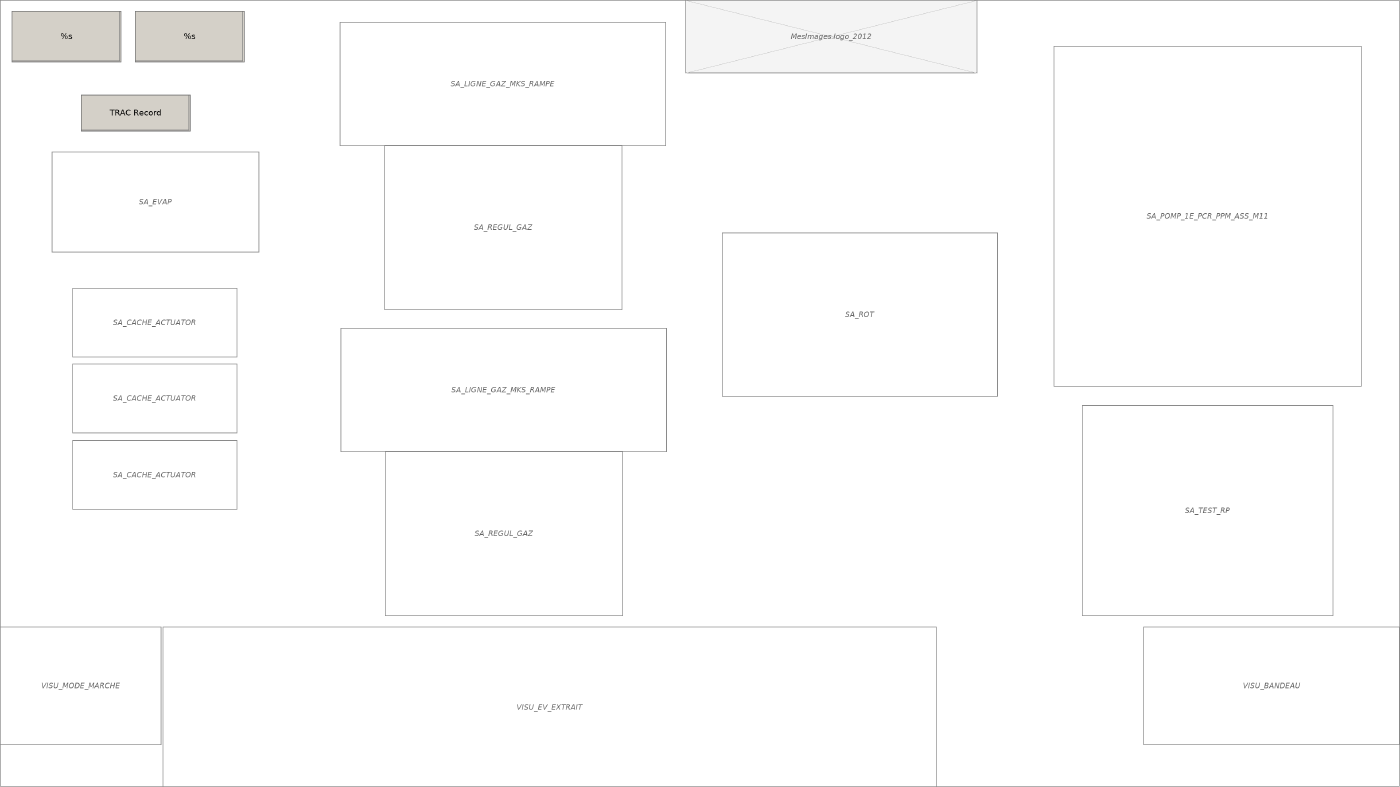
VISUALIZATION VISU_SA  // 1920x1080, background image fond_blanc_1280_1024
    Frame (223,860 1061x221)
        shows VISU_EV_EXTRAIT()
    Frame (1568,860 352x162)
        shows VISU_BANDEAU(m_Input_MACHINE := Global_Variables.MACHINE)
    Frame (0,860 221x162)
        shows VISU_MODE_MARCHE(m_Input_MACHINE := .MACHINE)
    Frame (71,208 284x138)
        shows SA_EVAP(m_Input_Crucible := PRG_EVAP.CRUCIBLE1, m_Input_Sweep := PRG_EVAP.SWEEP1)
    Frame (99,395 226x95)
        shows SA_CACHE_ACTUATOR(m_Input_CACHE := PRG_EVAP.CC11, m_Input_PRM_Forcage := PRG_EVAP.PRM_Forcage_Cache_Source1)
    Frame (466,30 447x170)
        shows SA_LIGNE_GAZ_MKS_RAMPE(m_Input_Ligne := PRG_GAZ.LIGNE_GAZ[1], m_Input_Machine := MACHINE, m_Input_DG := .PRG_GAZ.DG[1], m_Input_UserRight := PRG_USER.ACTU_USER.FONCTION_SA, m_Input_NumTextList := 11)
    Frame (99,499 226x95)
        shows SA_CACHE_ACTUATOR(m_Input_CACHE := PRG_EVAP.CC12, m_Input_PRM_Forcage := PRG_EVAP.PRM_Forcage_Cache_Source2)
    Frame (990,319 378x225)
        shows SA_ROT(m_Input_ROT := PRG_MOUVEMENT_PS.ROTATION_PS, m_Input_PRG := PRG_MOUVEMENT_PS)
    Frame (99,604 226x95)
        shows SA_CACHE_ACTUATOR(m_Input_CACHE := PRG_EVAP.CC13, m_Input_PRM_Forcage := PRG_EVAP.PRM_Forcage_Cache_Source3)
    Button (16,15 150x70), "%s", text list: 'TextList_Navigation', text index: 0
        OnMouseClick: change screen: SYN_POMPAGE
    Button (185,15 150x70), "%s", text list: 'TextList_Navigation', text index: 1
        OnMouseClick: change screen: SYN_PROC
    Frame (527,199 326x226)
        shows SA_REGUL_GAZ(m_Input_REGULATION := PRG_GAZ.REGULATION_GAZ_L1, m_Input_MACHINE := .MACHINE)
    Frame (528,619 326x226)
        shows SA_REGUL_GAZ(m_Input_REGULATION := PRG_GAZ.REGULATION_GAZ_L2, m_Input_MACHINE := .MACHINE)
    Frame (1484,556 344x289)
        shows SA_TEST_RP(m_Input_Operation := PRG_POMPAGE.POMPAGE.OP_Test_RP, m_Input_Pression := PRG_POMPAGE.POMPAGE.PRM_Pr_test, m_Input_Duree := PRG_POMPAGE.POMPAGE.PRM_Tim_test, m_Input_Volume := PRG_POMPAGE.POMPAGE.CONF_Volume_Enceinte, m_Input_Co_Stop := PRG_POMPAGE.POMPAGE.CO_Stop_Test_RP, m_Input_Timer := PRG_POMPAGE.POMPAGE.TIMER_attente_test.ET, m_Input_Result := PRG_POMPAGE.POMPAGE.VAR_Indicateur_Test)
    Frame (1445,63 422x467)
        shows SA_POMP_1E_PCR_PPM_ASS_M11(m_Input_PRG := PRG_POMPAGE, m_Input_Jauge := PRG_POMPAGE.M11, m_Input_Vanne := PRG_POMPAGE.POMPAGE.VS11, m_Input_Machine := MACHINE)
    Button (111,130 150x50), "TRAC Record", colour toggle: MAIN.Enr_TRAC
        toggle MAIN.Enr_TRAC
    Frame (467,450 447x170)
        shows SA_LIGNE_GAZ_MKS_RAMPE(m_Input_Ligne := PRG_GAZ.LIGNE_GAZ[2], m_Input_Machine := MACHINE, m_Input_DG := .PRG_GAZ.DG[2], m_Input_UserRight := PRG_USER.ACTU_USER.FONCTION_SA, m_Input_NumTextList := 12)
    Image (940,0 400x100), image: MesImages.logo_2012
END_VISUALIZATION

(* stored: Version 1.1.0.1, ProductVersion 3.1.4026.18
   Visu VISU_SA: Id {8a23c9c1-fb5e-4ae3-aaed-adcc3669ac75} *)
